{attribute 'qualified_only' := ''}
{attribute 'strict' := ''}
TYPE cStatus :
(
	None := 0,
	Empty := 1,
	Full := 2,
	RejectMalformedAPIData := 98,
	Reject := 99
) DINT;
END_TYPE

(* stored: Version 1.1.0.1, ProductVersion 3.1.4024.6
   DUT cStatus: Id {78b1cba2-157d-42ca-9498-c37202425431} *)
